PROGRAM MAIN
VAR
	Logger			: LogHelper<2>;
	LocalLog		: LocalLogger;
	initialized		: BOOL;
	Message			: LogMessage;
	Source			: LogSource;
	MotionArg		: MotionArgument;
	MotionParameters : ST_MotionParameters;
	
	//Commands
	logNoArgument	: BOOL;
	logWithArgument : BOOL;
END_VAR

IF NOT initialized THEN
	initialized			 := TRUE;
	MotionArg.Parameters REF= MotionParameters;
	Logger.Subscribe(LocalLog);
END_IF

IF logNoArgument THEN
	Source.SourceName := 'Test';
	Source.Timestamp := 123456789;
	Message.Message := 'Message';
	Message.Severity := 12;
	Logger.LogMessage(Source, Message);
	logNoArgument := FALSE;
END_IF

IF logWithArgument THEN
	Logger.LogMessage(Source, Message, MotionArg);
	logWithArgument := FALSE;
END_IF

END_PROGRAM

(* stored: Version 1.1.0.1, ProductVersion 3.1.4026.18
   POU MAIN: Id {c71f2366-b8c2-4cb7-b729-507396079bcf}, SpecialFunc None *)
